FUNCTION_BLOCK FB_AlarmHandler
VAR
END_VAR

METHOD Append : BOOL
VAR_INPUT
	tag : STRING;
	msg : STRING;
END_VAR
VAR
	str : STRING;
END_VAR
str := CONCAT(tag, ': ');
str := CONCAT(str, msg);
ADSLOGSTR(msgCtrlMask := ADSLOG_MSGTYPE_WARN OR ADSLOG_MSGTYPE_MSGBOX, msgFmtStr := '%s!', strArg := str);
END_METHOD

END_FUNCTION_BLOCK

(* stored: Version 1.1.0.1, ProductVersion 3.1.4024.11
   POU FB_AlarmHandler: Id {be54b949-3e78-4cf0-a2a1-cf3bd0f957b8}, SpecialFunc None
   Method Append: Id {10c19d97-2d21-49c7-a4e0-a87ea15bc7dd} *)
